// TIA Portal project "实验2_V20" (V20)

(* hardware
DEVICE "S7-300/ET200M station_1"  S7-300 station
   slot 0: "导轨_0"  Rail  6ES7 390-1***0-0AA0
   slot 2: "PLC_1"  CPU 314C-2 DP  6ES7 314-6CH04-0AB0  V3.3
      slot 0: "MPI 接口_1"  MPI
      slot 1: "DP 接口_1"  DP
      slot 2: "DI 24/DO 16_1"  DI24/DO16
      slot 3: "AI 5/AO 2_1"  AI5/AO2
      slot 4: "计数_1"  Counter
      slot 5: "定位_1"  Positioning
*)

// ===== PLC "PLC_1"  CPU 314C-2 DP =====

VAR_GLOBAL   // PLC tag table "默认变量表"
   "启动开关" AT %I0.0 : Bool;
   "运行状态" AT %M10.0 : Bool;
   "停止" AT %M10.1 : Bool;
   "手动" AT %I0.1 : Bool;
   "手动指示" AT %M10.2 : Bool;
   "速度1" AT %I0.2 : Bool;
   "速度2" AT %I0.3 : Bool;
   "速度3" AT %I0.4 : Bool;
   "正转" AT %I0.5 : Bool;
   "反转" AT %I0.6 : Bool;
   "单步" AT %I0.7 : Bool;
   "A相" AT %Q4.4 : Bool;
   "B相" AT %Q4.1 : Bool;
   "D相" AT %Q4.3 : Bool;
   "单步上升沿" AT %M10.4 : Bool;
   "按下单步的次数" AT %MW40 : Int;
   "C相" AT %Q4.2 : Bool;
   "速度1脉冲次数" AT %QW42 : Int;
   "速度2脉冲次数" AT %QW44 : Int;
   "速度3脉冲次数" AT %QW46 : Int;
   "速度1指示" AT %M10.3 : Bool;
   "速度2指示" AT %M10.5 : Bool;
   "速度3指示" AT %M10.6 : Bool;
END_VAR

DATA_BLOCK "速度模块_1_DB"   // DB2
{ S7_Optimized_Access := 'FALSE' }
VERSION : 0.1
// stored: InstanceOfName 速度模块_1
"速度模块_1"
BEGIN
END_DATA_BLOCK

FUNCTION_BLOCK "速度模块_1"   // FB1, LAD
{ S7_Optimized_Access := 'FALSE' }
VERSION : 0.1
BEGIN

REGION Network 1: 0.5Hz脉冲
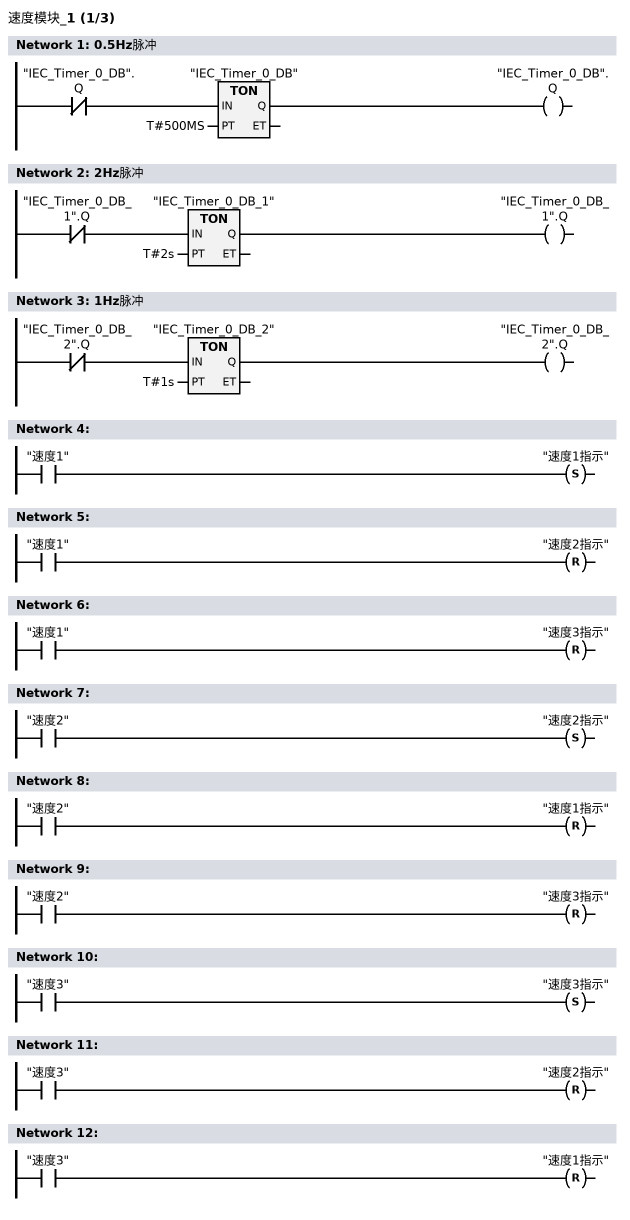
   "IEC_Timer_0_DB".TON(IN := NOT "IEC_Timer_0_DB".Q, PT := T#500MS);
   "IEC_Timer_0_DB".Q := "IEC_Timer_0_DB".Q;
END_REGION

REGION Network 2: 2Hz脉冲
   "IEC_Timer_0_DB_1".TON(IN := NOT "IEC_Timer_0_DB_1".Q, PT := T#2s);
   "IEC_Timer_0_DB_1".Q := "IEC_Timer_0_DB_1".Q;
END_REGION

REGION Network 3: 1Hz脉冲
   "IEC_Timer_0_DB_2".TON(IN := NOT "IEC_Timer_0_DB_2".Q, PT := T#1s);
   "IEC_Timer_0_DB_2".Q := "IEC_Timer_0_DB_2".Q;
END_REGION

REGION Network 4
   RUNG wire#powerrail
      Contact( "速度1" )
      S_Coil( "速度1指示" )
   END_RUNG
   // the same network as SCL:
   IF "速度1" THEN "速度1指示" := TRUE; END_IF;
END_REGION

REGION Network 5
   RUNG wire#powerrail
      Contact( "速度1" )
      R_Coil( "速度2指示" )
   END_RUNG
   // the same network as SCL:
   IF "速度1" THEN "速度2指示" := FALSE; END_IF;
END_REGION

REGION Network 6
   RUNG wire#powerrail
      Contact( "速度1" )
      R_Coil( "速度3指示" )
   END_RUNG
   // the same network as SCL:
   IF "速度1" THEN "速度3指示" := FALSE; END_IF;
END_REGION

REGION Network 7
   RUNG wire#powerrail
      Contact( "速度2" )
      S_Coil( "速度2指示" )
   END_RUNG
   // the same network as SCL:
   IF "速度2" THEN "速度2指示" := TRUE; END_IF;
END_REGION

REGION Network 8
   RUNG wire#powerrail
      Contact( "速度2" )
      R_Coil( "速度1指示" )
   END_RUNG
   // the same network as SCL:
   IF "速度2" THEN "速度1指示" := FALSE; END_IF;
END_REGION

REGION Network 9
   RUNG wire#powerrail
      Contact( "速度2" )
      R_Coil( "速度3指示" )
   END_RUNG
   // the same network as SCL:
   IF "速度2" THEN "速度3指示" := FALSE; END_IF;
END_REGION

REGION Network 10
   RUNG wire#powerrail
      Contact( "速度3" )
      S_Coil( "速度3指示" )
   END_RUNG
   // the same network as SCL:
   IF "速度3" THEN "速度3指示" := TRUE; END_IF;
END_REGION

REGION Network 11
   RUNG wire#powerrail
      Contact( "速度3" )
      R_Coil( "速度2指示" )
   END_RUNG
   // the same network as SCL:
   IF "速度3" THEN "速度2指示" := FALSE; END_IF;
END_REGION

REGION Network 12
   RUNG wire#powerrail
      Contact( "速度3" )
      R_Coil( "速度1指示" )
   END_RUNG
   // the same network as SCL:
   IF "速度3" THEN "速度1指示" := FALSE; END_IF;
END_REGION

REGION Network 13
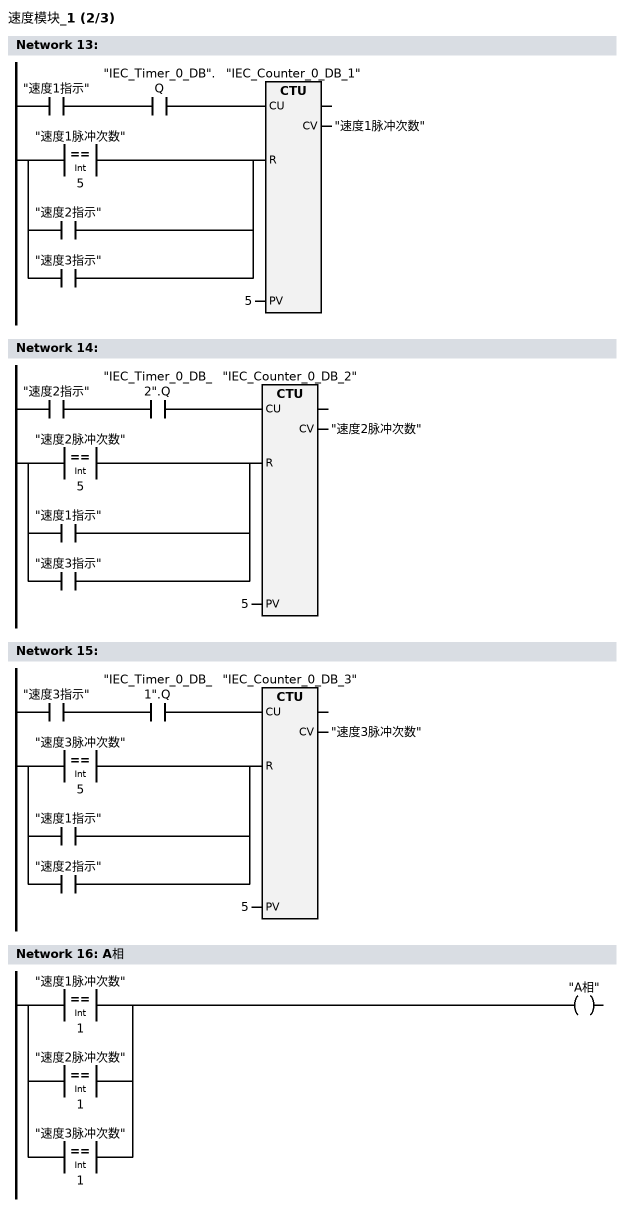
   "IEC_Counter_0_DB_1".CTU(CU := "速度1指示" AND "IEC_Timer_0_DB".Q,
                           R := ("速度1脉冲次数" = 5) OR "速度2指示" OR "速度3指示",
                           PV := 5,
                           CV => "速度1脉冲次数");
END_REGION

REGION Network 14
   "IEC_Counter_0_DB_2".CTU(CU := "速度2指示" AND "IEC_Timer_0_DB_2".Q,
                           R := ("速度2脉冲次数" = 5) OR "速度1指示" OR "速度3指示",
                           PV := 5,
                           CV => "速度2脉冲次数");
END_REGION

REGION Network 15
   "IEC_Counter_0_DB_3".CTU(CU := "速度3指示" AND "IEC_Timer_0_DB_1".Q,
                           R := ("速度3脉冲次数" = 5) OR "速度1指示" OR "速度2指示",
                           PV := 5,
                           CV => "速度3脉冲次数");
END_REGION

REGION Network 16: A相
   RUNG wire#powerrail
      { S7_Templates := "SrcType := Int" } EQ_Contact(in1 := "速度1脉冲次数", in2 := 1)
      wire#w1
      Coil( "A相" )
   END_RUNG
   RUNG wire#powerrail
      { S7_Templates := "SrcType := Int" } EQ_Contact(in1 := "速度2脉冲次数", in2 := 1)
   END_RUNG wire#w1
   RUNG wire#powerrail
      { S7_Templates := "SrcType := Int" } EQ_Contact(in1 := "速度3脉冲次数", in2 := 1)
   END_RUNG wire#w1
   // the same network as SCL:
   "A相" := ("速度1脉冲次数" = 1) OR ("速度2脉冲次数" = 1) OR ("速度3脉冲次数" = 1);
END_REGION

REGION Network 17: B相
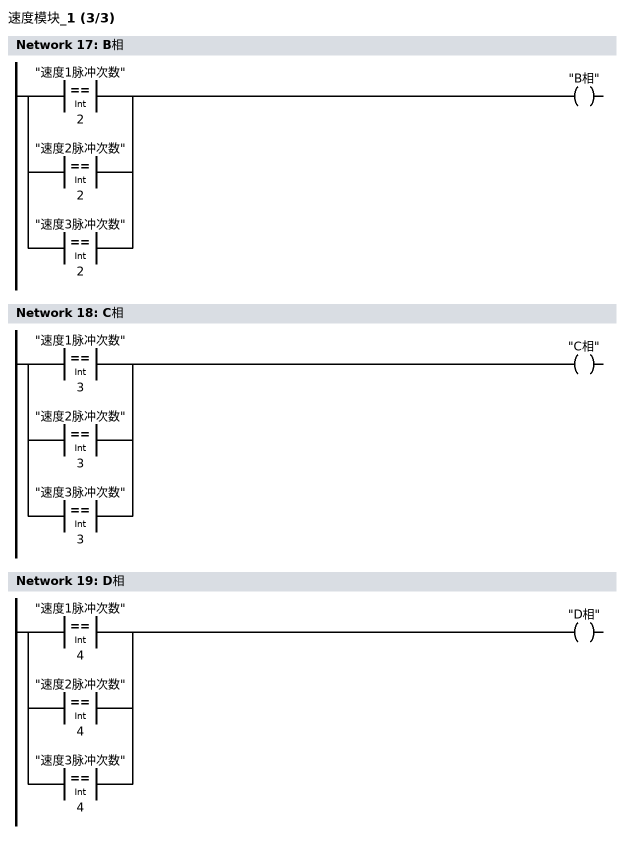
   RUNG wire#powerrail
      { S7_Templates := "SrcType := Int" } EQ_Contact(in1 := "速度1脉冲次数", in2 := 2)
      wire#w1
      Coil( "B相" )
   END_RUNG
   RUNG wire#powerrail
      { S7_Templates := "SrcType := Int" } EQ_Contact(in1 := "速度2脉冲次数", in2 := 2)
   END_RUNG wire#w1
   RUNG wire#powerrail
      { S7_Templates := "SrcType := Int" } EQ_Contact(in1 := "速度3脉冲次数", in2 := 2)
   END_RUNG wire#w1
   // the same network as SCL:
   "B相" := ("速度1脉冲次数" = 2) OR ("速度2脉冲次数" = 2) OR ("速度3脉冲次数" = 2);
END_REGION

REGION Network 18: C相
   RUNG wire#powerrail
      { S7_Templates := "SrcType := Int" } EQ_Contact(in1 := "速度1脉冲次数", in2 := 3)
      wire#w1
      Coil( "C相" )
   END_RUNG
   RUNG wire#powerrail
      { S7_Templates := "SrcType := Int" } EQ_Contact(in1 := "速度2脉冲次数", in2 := 3)
   END_RUNG wire#w1
   RUNG wire#powerrail
      { S7_Templates := "SrcType := Int" } EQ_Contact(in1 := "速度3脉冲次数", in2 := 3)
   END_RUNG wire#w1
   // the same network as SCL:
   "C相" := ("速度1脉冲次数" = 3) OR ("速度2脉冲次数" = 3) OR ("速度3脉冲次数" = 3);
END_REGION

REGION Network 19: D相
   RUNG wire#powerrail
      { S7_Templates := "SrcType := Int" } EQ_Contact(in1 := "速度1脉冲次数", in2 := 4)
      wire#w1
      Coil( "D相" )
   END_RUNG
   RUNG wire#powerrail
      { S7_Templates := "SrcType := Int" } EQ_Contact(in1 := "速度2脉冲次数", in2 := 4)
   END_RUNG wire#w1
   RUNG wire#powerrail
      { S7_Templates := "SrcType := Int" } EQ_Contact(in1 := "速度3脉冲次数", in2 := 4)
   END_RUNG wire#w1
   // the same network as SCL:
   "D相" := ("速度1脉冲次数" = 4) OR ("速度2脉冲次数" = 4) OR ("速度3脉冲次数" = 4);
END_REGION
END_FUNCTION_BLOCK

ORGANIZATION_BLOCK "Main"   // OB1, LAD
TITLE = "Main Program Sweep (Cycle)"
{ S7_Optimized_Access := 'FALSE' }
VERSION : 0.1
   VAR_TEMP
      OB1_EV_CLASS : Byte;   // Bits 0-3 = 1 (Coming event), Bits 4-7 = 1 (Event class 1)
      OB1_SCAN_1 : Byte;   // 1 (Cold restart scan 1 of OB 1), 3 (Scan 2-n of OB 1)
      OB1_PRIORITY : Byte;   // Priority of OB Execution
      OB1_OB_NUMBR : Byte;   // 1 (Organization block 1, OB1)
      OB1_RESERVED_1 : Byte;   // Reserved for system
      OB1_RESERVED_2 : Byte;   // Reserved for system
      OB1_PREV_CYCLE : Int;   // Cycle time of previous OB1 scan (milliseconds)
      OB1_MIN_CYCLE : Int;   // Minimum cycle time of OB1 (milliseconds)
      OB1_MAX_CYCLE : Int;   // Maximum cycle time of OB1 (milliseconds)
      OB1_DATE_TIME : Date_And_Time;   // Date and time OB1 started
   END_VAR
   VAR_TEMP   // added for the SCL form of the ladder/FBD networks
      _w1 : Bool;
   END_VAR
BEGIN

REGION Network 1
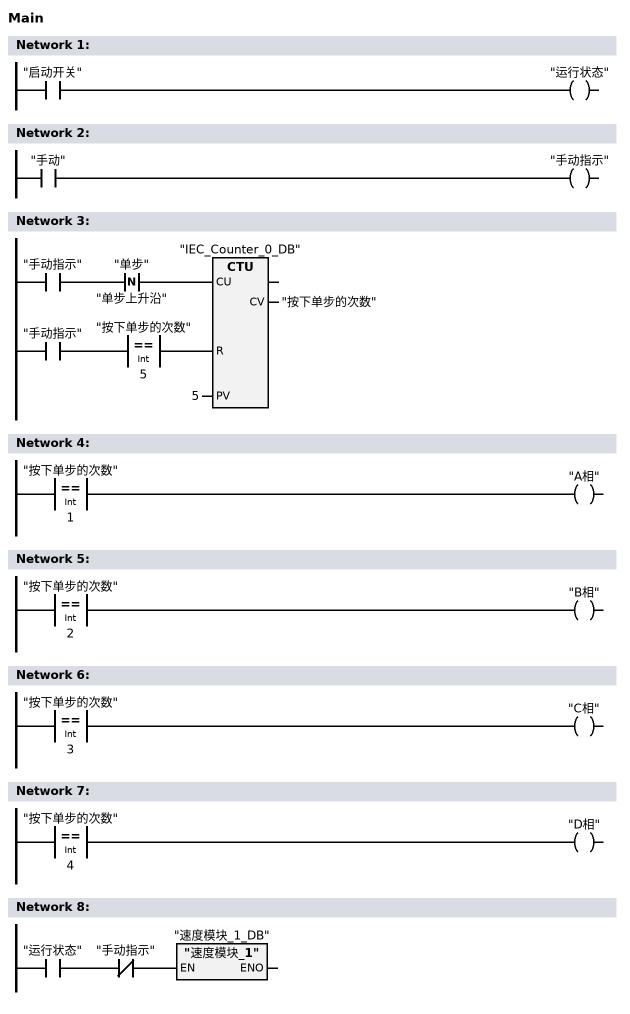
   RUNG wire#powerrail
      Contact( "启动开关" )
      Coil( "运行状态" )
   END_RUNG
   // the same network as SCL:
   "运行状态" := "启动开关";
END_REGION

REGION Network 2
   RUNG wire#powerrail
      Contact( "手动" )
      Coil( "手动指示" )
   END_RUNG
   // the same network as SCL:
   "手动指示" := "手动";
END_REGION

REGION Network 3
   #_w1 := "手动指示" AND NOT "单步" AND "单步上升沿";   // falling edge of "单步"
   "单步上升沿" := "单步";
   "IEC_Counter_0_DB".CTU(CU := #_w1, R := "手动指示" AND ("按下单步的次数" = 5), PV := 5, CV => "按下单步的次数");
END_REGION

REGION Network 4
   RUNG wire#powerrail
      { S7_Templates := "SrcType := Int" } EQ_Contact(in1 := "按下单步的次数", in2 := 1)
      Coil( "A相" )
   END_RUNG
   // the same network as SCL:
   "A相" := "按下单步的次数" = 1;
END_REGION

REGION Network 5
   RUNG wire#powerrail
      { S7_Templates := "SrcType := Int" } EQ_Contact(in1 := "按下单步的次数", in2 := 2)
      Coil( "B相" )
   END_RUNG
   // the same network as SCL:
   "B相" := "按下单步的次数" = 2;
END_REGION

REGION Network 6
   RUNG wire#powerrail
      { S7_Templates := "SrcType := Int" } EQ_Contact(in1 := "按下单步的次数", in2 := 3)
      Coil( "C相" )
   END_RUNG
   // the same network as SCL:
   "C相" := "按下单步的次数" = 3;
END_REGION

REGION Network 7
   RUNG wire#powerrail
      { S7_Templates := "SrcType := Int" } EQ_Contact(in1 := "按下单步的次数", in2 := 4)
      Coil( "D相" )
   END_RUNG
   // the same network as SCL:
   "D相" := "按下单步的次数" = 4;
END_REGION

REGION Network 8
   RUNG wire#powerrail
      Contact( "运行状态" )
      I_Contact( "手动指示" )
      "速度模块_1_DB"()
   END_RUNG
   // the same network as SCL:
   IF "运行状态" AND NOT "手动指示" THEN
       "速度模块_1_DB"();   // "速度模块_1"
   END_IF;
END_REGION
END_ORGANIZATION_BLOCK